// =============================================================================
// 02b_RecipePrograms.scl
// Recipe program data blocks (DB_RecipeProgram1..10)
//
// *** GENERATED FILE -- do not hand-edit. ***
// Produced by tools/gen_recipe_slots.py --slots 10
// To change the slot count, run that script; do not add declarations by hand.
//
// Kept separate from 02_DataBlocks.scl so real recipe data is not overwritten
// when 02_DataBlocks.scl is regenerated.
// Depends on: 01_DataTypes.scl (RecipeHeader, RecipeLine UDTs)
//
// *** IMPORTING THIS FILE INTO TIA WIPES ALL RECIPE DATA ***
// (warning added 2026-08-06, field commissioning)
// The BEGIN blocks below are EMPTY -- these declarations exist only so the
// project compiles before any CAM file arrives. The real recipe data lives in
// the CAM-generated files (gcodes/DB_RecipeProgramN.scl), which declare the
// SAME block names and overwrite these when imported. Importing THIS file after
// a CAM import therefore replaces every recipe with all-zero data -- and because
// the DBs are UNLINKED (load memory only, not monitorable online), the wipe is
// invisible until a cycle start copies zeros into DB_SelectedRecipe. Pre-scan
// catches that as 16#0313 (missing END marker), but the recipes are still gone.
//
// So the import order is not optional:
//     1. this file        (structure)
//     2. EVERY gcodes/DB_RecipeProgramN.scl   (data)
// Never step 1 without step 2.
//
// =============================================================================
// LOAD-MEMORY RECIPES (2026-08-04) -- read this before editing the generator
// =============================================================================
// These DBs live in LOAD MEMORY ONLY. They cost zero work memory. FB_Process
// copies the selected one into "DB_SelectedRecipe" (work memory) with READ_DBL
// in STATE_RECIPE_LOAD(11), and everything downstream runs from that buffer.
// Design + gate-test evidence: Program/docs/LOADMEM_COPY_ON_SELECT.md
//
// THREE THINGS THE CAM POST-PROCESSOR MUST EMIT, EXACTLY:
//
//   1. { S7_Optimized_Access := 'FALSE' }   -- standard access.
//      READ_DBL requires source and destination to have the SAME access type,
//      and an optimized DB may not contain a STRUCT (RecipeLine is a UDT).
//      An optimized recipe DB is REFUSED by READ_DBL at runtime.
//
//   2. UNLINKED  -- and it MUST come BEFORE NON_RETAIN.
//      Verified on TIA V17 / S7-1214C 2026-08-04: NON_RETAIN then UNLINKED
//      will NOT generate blocks from the source. The order below is the one
//      that works.
//
//      *** OMITTING UNLINKED FAILS SILENTLY. ***
//      The recipe then sits in work memory, READ_DBL still succeeds (it reads
//      the DB's start values either way), every test still passes, and the
//      only symptom is that ~9 KB of work memory per recipe is quietly
//      consumed again. It will not surface until the CPU runs out. Wrong
//      ORDER is loud (nothing generates); a MISSING line is silent.
//
//   3. Array[0..799] -- 800 lines. Must match DB_SelectedRecipe exactly.
//      Header.LineCount is validated against 1..800 in STATE_PRE_SCAN(12).
//
// A load-memory-only DB CANNOT be monitored online -- that is expected, and is
// the quickest proof the attribute took effect. To inspect recipe data, run a
// cycle and look at DB_SelectedRecipe instead.
//
// Slot count does NOT affect scan time: FB_RecipeLoader's CASE executes exactly
// one branch per scan regardless of how many slots exist, and unselected recipes
// are never touched.
//
// It DOES cost work memory, which is the constraint that bites. These DBs are free
// (UNLINKED, load memory), but the loader CASE is two READ_DBL call sites per slot
// and on the S7-1200 compiled code lives in the same 100 KB work memory as the DB
// data. 50 slots compiled to 101% on 2026-08-10 and would not download.
//
// *** THE COUNT HERE MAY DELIBERATELY EXCEED THE LOADER'S COUNT. ***
// FB_RecipeLoader's PROGRAM_COUNT and the activeProgram clamp may be LOWER than
// the number of DATA_BLOCKs below, while the work-memory budget is being tuned
// with gen_recipe_slots.py --loader-only. Surplus declarations are harmless: they
// cost load memory (plenty spare) and the clamp makes them unreachable. The
// LOADER's count is the number of slots an operator can actually select -- not the
// number of DATA_BLOCKs in this file. The generator refuses to shrink this file
// without --shrink-02b, because importing a shrunk 02b wipes recipe data as well
// as removing declarations.
//
// Load memory cost: 10 x ~9 KB = ~0.09 MB of the 1214C's 4 MB.
// =============================================================================

// -----------------------------------------------------------------------------
// DB_RecipeChunk - staging area for ONE chunk of a recipe (100 lines)
//
// Chunked transfer (2026-08-13): a single 12 KB READ_DBL out of load memory
// lands only partially on this CPU, with RET_VAL = 0 and no error. Each chunk is
// now pulled into this buffer, verified line by line, and only then copied into
// DB_SelectedRecipe. 100 lines is small enough that EVERY line can be
// checked rather than sampled -- there is no hole this can miss.
//
// Cost: 1200 bytes of work memory, once, regardless of slot count.
// -----------------------------------------------------------------------------
DATA_BLOCK "DB_RecipeChunk"
{ S7_Optimized_Access := 'FALSE' }
VERSION : 0.1
NON_RETAIN
    VAR
        Lines : Array[0..99] of "RecipeLine";
    END_VAR
BEGIN
END_DATA_BLOCK

// -----------------------------------------------------------------------------
// DB_RecipeProgram1 - Recipe data for Program 1
// -----------------------------------------------------------------------------
DATA_BLOCK "DB_RecipeProgram1"
{ S7_Optimized_Access := 'FALSE' }
VERSION : 0.3
UNLINKED
NON_RETAIN
    VAR
        Header : "RecipeHeader";                // Program name, LineCount, Valid, bounding box, tool table
        Lines1 : Array[0..99] of "RecipeLine"; // global lines 0..99
        Lines2 : Array[0..99] of "RecipeLine"; // global lines 100..199
        Lines3 : Array[0..99] of "RecipeLine"; // global lines 200..299
        Lines4 : Array[0..99] of "RecipeLine"; // global lines 300..399
        Lines5 : Array[0..99] of "RecipeLine"; // global lines 400..499
        Lines6 : Array[0..99] of "RecipeLine"; // global lines 500..599
        Lines7 : Array[0..99] of "RecipeLine"; // global lines 600..699
        Lines8 : Array[0..99] of "RecipeLine"; // global lines 700..799
    END_VAR
BEGIN
END_DATA_BLOCK

// -----------------------------------------------------------------------------
// DB_RecipeProgram2 - Recipe data for Program 2
// -----------------------------------------------------------------------------
DATA_BLOCK "DB_RecipeProgram2"
{ S7_Optimized_Access := 'FALSE' }
VERSION : 0.3
UNLINKED
NON_RETAIN
    VAR
        Header : "RecipeHeader";                // Program name, LineCount, Valid, bounding box, tool table
        Lines1 : Array[0..99] of "RecipeLine"; // global lines 0..99
        Lines2 : Array[0..99] of "RecipeLine"; // global lines 100..199
        Lines3 : Array[0..99] of "RecipeLine"; // global lines 200..299
        Lines4 : Array[0..99] of "RecipeLine"; // global lines 300..399
        Lines5 : Array[0..99] of "RecipeLine"; // global lines 400..499
        Lines6 : Array[0..99] of "RecipeLine"; // global lines 500..599
        Lines7 : Array[0..99] of "RecipeLine"; // global lines 600..699
        Lines8 : Array[0..99] of "RecipeLine"; // global lines 700..799
    END_VAR
BEGIN
END_DATA_BLOCK

// -----------------------------------------------------------------------------
// DB_RecipeProgram3 - Recipe data for Program 3
// -----------------------------------------------------------------------------
DATA_BLOCK "DB_RecipeProgram3"
{ S7_Optimized_Access := 'FALSE' }
VERSION : 0.3
UNLINKED
NON_RETAIN
    VAR
        Header : "RecipeHeader";                // Program name, LineCount, Valid, bounding box, tool table
        Lines1 : Array[0..99] of "RecipeLine"; // global lines 0..99
        Lines2 : Array[0..99] of "RecipeLine"; // global lines 100..199
        Lines3 : Array[0..99] of "RecipeLine"; // global lines 200..299
        Lines4 : Array[0..99] of "RecipeLine"; // global lines 300..399
        Lines5 : Array[0..99] of "RecipeLine"; // global lines 400..499
        Lines6 : Array[0..99] of "RecipeLine"; // global lines 500..599
        Lines7 : Array[0..99] of "RecipeLine"; // global lines 600..699
        Lines8 : Array[0..99] of "RecipeLine"; // global lines 700..799
    END_VAR
BEGIN
END_DATA_BLOCK

// -----------------------------------------------------------------------------
// DB_RecipeProgram4 - Recipe data for Program 4
// -----------------------------------------------------------------------------
DATA_BLOCK "DB_RecipeProgram4"
{ S7_Optimized_Access := 'FALSE' }
VERSION : 0.3
UNLINKED
NON_RETAIN
    VAR
        Header : "RecipeHeader";                // Program name, LineCount, Valid, bounding box, tool table
        Lines1 : Array[0..99] of "RecipeLine"; // global lines 0..99
        Lines2 : Array[0..99] of "RecipeLine"; // global lines 100..199
        Lines3 : Array[0..99] of "RecipeLine"; // global lines 200..299
        Lines4 : Array[0..99] of "RecipeLine"; // global lines 300..399
        Lines5 : Array[0..99] of "RecipeLine"; // global lines 400..499
        Lines6 : Array[0..99] of "RecipeLine"; // global lines 500..599
        Lines7 : Array[0..99] of "RecipeLine"; // global lines 600..699
        Lines8 : Array[0..99] of "RecipeLine"; // global lines 700..799
    END_VAR
BEGIN
END_DATA_BLOCK

// -----------------------------------------------------------------------------
// DB_RecipeProgram5 - Recipe data for Program 5
// -----------------------------------------------------------------------------
DATA_BLOCK "DB_RecipeProgram5"
{ S7_Optimized_Access := 'FALSE' }
VERSION : 0.3
UNLINKED
NON_RETAIN
    VAR
        Header : "RecipeHeader";                // Program name, LineCount, Valid, bounding box, tool table
        Lines1 : Array[0..99] of "RecipeLine"; // global lines 0..99
        Lines2 : Array[0..99] of "RecipeLine"; // global lines 100..199
        Lines3 : Array[0..99] of "RecipeLine"; // global lines 200..299
        Lines4 : Array[0..99] of "RecipeLine"; // global lines 300..399
        Lines5 : Array[0..99] of "RecipeLine"; // global lines 400..499
        Lines6 : Array[0..99] of "RecipeLine"; // global lines 500..599
        Lines7 : Array[0..99] of "RecipeLine"; // global lines 600..699
        Lines8 : Array[0..99] of "RecipeLine"; // global lines 700..799
    END_VAR
BEGIN
END_DATA_BLOCK

// -----------------------------------------------------------------------------
// DB_RecipeProgram6 - Recipe data for Program 6
// -----------------------------------------------------------------------------
DATA_BLOCK "DB_RecipeProgram6"
{ S7_Optimized_Access := 'FALSE' }
VERSION : 0.3
UNLINKED
NON_RETAIN
    VAR
        Header : "RecipeHeader";                // Program name, LineCount, Valid, bounding box, tool table
        Lines1 : Array[0..99] of "RecipeLine"; // global lines 0..99
        Lines2 : Array[0..99] of "RecipeLine"; // global lines 100..199
        Lines3 : Array[0..99] of "RecipeLine"; // global lines 200..299
        Lines4 : Array[0..99] of "RecipeLine"; // global lines 300..399
        Lines5 : Array[0..99] of "RecipeLine"; // global lines 400..499
        Lines6 : Array[0..99] of "RecipeLine"; // global lines 500..599
        Lines7 : Array[0..99] of "RecipeLine"; // global lines 600..699
        Lines8 : Array[0..99] of "RecipeLine"; // global lines 700..799
    END_VAR
BEGIN
END_DATA_BLOCK

// -----------------------------------------------------------------------------
// DB_RecipeProgram7 - Recipe data for Program 7
// -----------------------------------------------------------------------------
DATA_BLOCK "DB_RecipeProgram7"
{ S7_Optimized_Access := 'FALSE' }
VERSION : 0.3
UNLINKED
NON_RETAIN
    VAR
        Header : "RecipeHeader";                // Program name, LineCount, Valid, bounding box, tool table
        Lines1 : Array[0..99] of "RecipeLine"; // global lines 0..99
        Lines2 : Array[0..99] of "RecipeLine"; // global lines 100..199
        Lines3 : Array[0..99] of "RecipeLine"; // global lines 200..299
        Lines4 : Array[0..99] of "RecipeLine"; // global lines 300..399
        Lines5 : Array[0..99] of "RecipeLine"; // global lines 400..499
        Lines6 : Array[0..99] of "RecipeLine"; // global lines 500..599
        Lines7 : Array[0..99] of "RecipeLine"; // global lines 600..699
        Lines8 : Array[0..99] of "RecipeLine"; // global lines 700..799
    END_VAR
BEGIN
END_DATA_BLOCK

// -----------------------------------------------------------------------------
// DB_RecipeProgram8 - Recipe data for Program 8
// -----------------------------------------------------------------------------
DATA_BLOCK "DB_RecipeProgram8"
{ S7_Optimized_Access := 'FALSE' }
VERSION : 0.3
UNLINKED
NON_RETAIN
    VAR
        Header : "RecipeHeader";                // Program name, LineCount, Valid, bounding box, tool table
        Lines1 : Array[0..99] of "RecipeLine"; // global lines 0..99
        Lines2 : Array[0..99] of "RecipeLine"; // global lines 100..199
        Lines3 : Array[0..99] of "RecipeLine"; // global lines 200..299
        Lines4 : Array[0..99] of "RecipeLine"; // global lines 300..399
        Lines5 : Array[0..99] of "RecipeLine"; // global lines 400..499
        Lines6 : Array[0..99] of "RecipeLine"; // global lines 500..599
        Lines7 : Array[0..99] of "RecipeLine"; // global lines 600..699
        Lines8 : Array[0..99] of "RecipeLine"; // global lines 700..799
    END_VAR
BEGIN
END_DATA_BLOCK

// -----------------------------------------------------------------------------
// DB_RecipeProgram9 - Recipe data for Program 9
// -----------------------------------------------------------------------------
DATA_BLOCK "DB_RecipeProgram9"
{ S7_Optimized_Access := 'FALSE' }
VERSION : 0.3
UNLINKED
NON_RETAIN
    VAR
        Header : "RecipeHeader";                // Program name, LineCount, Valid, bounding box, tool table
        Lines1 : Array[0..99] of "RecipeLine"; // global lines 0..99
        Lines2 : Array[0..99] of "RecipeLine"; // global lines 100..199
        Lines3 : Array[0..99] of "RecipeLine"; // global lines 200..299
        Lines4 : Array[0..99] of "RecipeLine"; // global lines 300..399
        Lines5 : Array[0..99] of "RecipeLine"; // global lines 400..499
        Lines6 : Array[0..99] of "RecipeLine"; // global lines 500..599
        Lines7 : Array[0..99] of "RecipeLine"; // global lines 600..699
        Lines8 : Array[0..99] of "RecipeLine"; // global lines 700..799
    END_VAR
BEGIN
END_DATA_BLOCK

// -----------------------------------------------------------------------------
// DB_RecipeProgram10 - Recipe data for Program 10
// -----------------------------------------------------------------------------
DATA_BLOCK "DB_RecipeProgram10"
{ S7_Optimized_Access := 'FALSE' }
VERSION : 0.3
UNLINKED
NON_RETAIN
    VAR
        Header : "RecipeHeader";                // Program name, LineCount, Valid, bounding box, tool table
        Lines1 : Array[0..99] of "RecipeLine"; // global lines 0..99
        Lines2 : Array[0..99] of "RecipeLine"; // global lines 100..199
        Lines3 : Array[0..99] of "RecipeLine"; // global lines 200..299
        Lines4 : Array[0..99] of "RecipeLine"; // global lines 300..399
        Lines5 : Array[0..99] of "RecipeLine"; // global lines 400..499
        Lines6 : Array[0..99] of "RecipeLine"; // global lines 500..599
        Lines7 : Array[0..99] of "RecipeLine"; // global lines 600..699
        Lines8 : Array[0..99] of "RecipeLine"; // global lines 700..799
    END_VAR
BEGIN
END_DATA_BLOCK
